TYPE TupleStruct_2:
    STRUCT
        field0: BOOL;
        field1: DINT;
        field2: LREAL;
    END_STRUCT;
END_TYPE
